// TwinCAT 3 PLC project Este_es_el_PLC
// ProgramVersion: 3.1.4024.0
// libraries:
//   Tc2_EtherCAT, * (Beckhoff Automation GmbH)
//   Tc2_ModbusSrv, * (Beckhoff Automation GmbH)
//   Tc2_Standard, * (Beckhoff Automation GmbH)
//   Tc2_System, * (Beckhoff Automation GmbH)
//   Tc2_Utilities, * (Beckhoff Automation GmbH)
//   Tc3_Module, * (Beckhoff Automation GmbH)
// project tree:
//   DUTs/ E_EventType.TcDUT (not stored), St_Event.TcDUT (not stored), ST_MachineStation.TcDUT
//   GVLs/ GVL.TcGVL (not stored), Tags.TcGVL (not stored)
//   / PlcTask.TcTTO (not stored)
//   POUs/ conveyor1.TcPOU (not stored), MAIN.TcPOU
// real-time tasks:
//   TASK PlcTask: cycle T#10ms, priority 20, ADS port 350
//   TASK Device 1 (OPC UA Virtual)_Task_58: cycle T#40ms, priority 58, ADS port 351

// ---- DUTs/ST_MachineStation.TcDUT
TYPE ST_MachineStation :
STRUCT
	iSensorInfeed1, 		
	iSensorInfeed2, 		
	iSensorOutfeed1, 	
	iSensorOutfeed2, 	
	bButtonMachineStart,
	bButtonMachineStop,
	bButtonMachineReset : BOOL;
			
END_STRUCT
END_TYPE

// ---- POUs/MAIN.TcPOU
PROGRAM MAIN
VAR
	bButtonStart,
	bButtonReset,
	bButtonStop: BOOL;
	bStatus : BOOL;
	bButtonLightStart,
	bButtonLightStop,
	bExtra, botroextra,bTercer : BOOL;
END_VAR

bButtonStart := GVL.mb_Output_Coils[0];
bButtonStop := GVL.mb_Output_Coils[1];
bButtonReset := GVL.mb_Output_Coils[29];
GVL.mb_Input_Coils[0] := bButtonLightStart;
GVL.mb_Input_Coils[1] := bButtonLightStop;
conveyor1();

Tags.bAutoMan(SET1 := bButtonStart, RESET := NOT bButtonStop);
bStatus := Tags.bAutoMan.Q1;
bButtonLightStart := bStatus;
bButtonLightStop := not bStatus;

END_PROGRAM
